Fanuc KAREL source: kt00087.compact.KL

PROGRAM KT00087
%STACKSIZE=65535
%PRIORITY=65535
%NOLOCKGROUP
VAR
Y1 : ARRAY[2] OF BYTE
H2 : ARRAY[2] OF SHORT
OUT : INTEGER
BEGIN
Y1[1]=2
H2[1]=3
OUT=(Y1[1] * H2[1])
END KT00087
